(* Logix 5000 project; controller Lab7_1 5069-L306ERM rev 35.16; software revision 35.00 *)

TASK MainTask (continuous, watchdog 500 ms) : MainProgram

MODULES
   Local : 5069-L306ERM (5069 0, rev 35.16)
      IOHub : vendor 1 type 7 code 358 (Ethernet 192.168.110.5, rev 1.1, Output RPI 20 ms)
END_MODULES

PROGRAM MainProgram   (* main routine MainRoutine *)
VAR
   countDown2 : COUNTER := (PRE := 2);
   countDown3 : COUNTER := (PRE := 3);
   counter_0 : COUNTER;
   counter_2 : COUNTER;
   displayTimer : TIMER := (PRE := 5000);
   Dummy : BOOL;
   enable_1_sec : BOOL;
   enable_3_sec : BOOL;
   flash1 : BOOL;
   flash1TOF : TIMER := (PRE := 500);
   flash2 : BOOL;
   flash2TOF : TIMER := (PRE := 1000);
   flash2TON : TIMER := (PRE := 1000);
   flash3 : BOOL;
   flash3TOF : TIMER := (PRE := 1000);
   flash3TON : TIMER := (PRE := 1000);
   flash_1 : BOOL;
   flash_1TOF : TIMER := (PRE := 1000);
   flash_2 : BOOL;
   flash_3 : BOOL;
   HOLD : BOOL;
   HOLD2 : BOOL;
   light_test : BOOL;
   reset : BOOL;
   timer : TIMER := (PRE := 999999999);
   timer_1 : TIMER := (PRE := 1000);
   timer_1_delay : TIMER := (PRE := 1000);
   timer_1_sec : TIMER := (PRE := 1000);
   timer_2 : TIMER := (PRE := 1000);
   timer_2_1 : TIMER := (PRE := 2000);
   timer_2_delay : TIMER := (PRE := 3000, ACC := 2000);
   timer_3_1 : TIMER := (PRE := 3000);
   timer_3_delay : TIMER := (PRE := 5000);
   timer_3_sec : TIMER := (PRE := 1000);
   timer_flash_1 : TIMER := (PRE := 2000);
   timer_flash_2 : TIMER := (PRE := 4000);
   timer_flash_3 : TIMER := (PRE := 6000);
END_VAR

ROUTINE MainRoutine   (* ladder *)
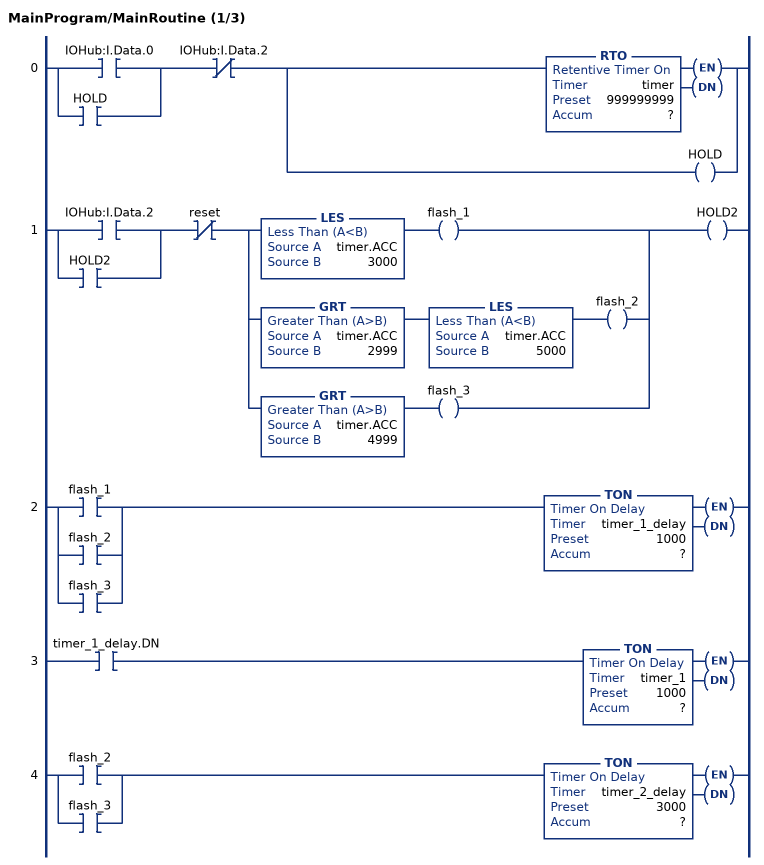
   0: [XIC(IOHub:I.Data.0) ,XIC(HOLD) ]XIO(IOHub:I.Data.2)[RTO(timer,?,?) ,OTE(HOLD) ];
   1: [XIC(IOHub:I.Data.2) ,XIC(HOLD2) ]XIO(reset)[LES(timer.ACC,3000) OTE(flash_1) ,[GRT(timer.ACC,2999) LES(timer.ACC,5000) OTE(flash_2) ,GRT(timer.ACC,4999) OTE(flash_3) ] ]OTE(HOLD2);
   2: [XIC(flash_1) ,XIC(flash_2) ,XIC(flash_3) ]TON(timer_1_delay,?,?);
   3: XIC(timer_1_delay.DN)TON(timer_1,?,?);
   4: [XIC(flash_2) ,XIC(flash_3) ]TON(timer_2_delay,?,?);
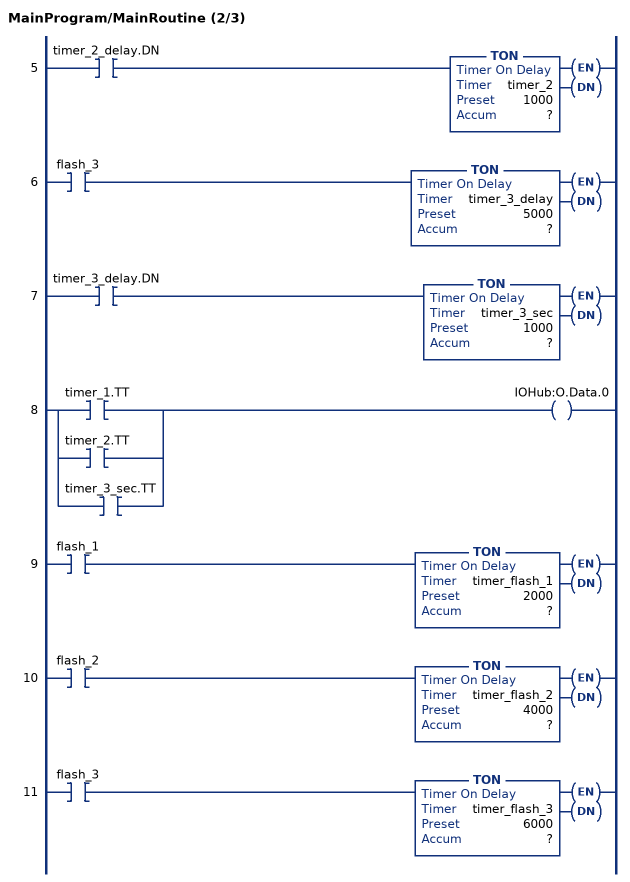
   5: XIC(timer_2_delay.DN)TON(timer_2,?,?);
   6: XIC(flash_3)TON(timer_3_delay,?,?);
   7: XIC(timer_3_delay.DN)TON(timer_3_sec,?,?);
   8: [XIC(timer_1.TT) ,[XIC(timer_2.TT) ,XIC(timer_3_sec.TT) ] ]OTE(IOHub:O.Data.0);
   9: XIC(flash_1)TON(timer_flash_1,?,?);
   10: XIC(flash_2)TON(timer_flash_2,?,?);
   11: XIC(flash_3)TON(timer_flash_3,?,?);
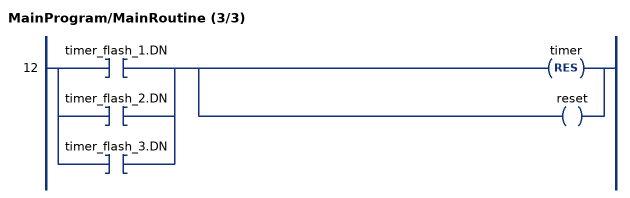
   12: [XIC(timer_flash_1.DN) ,XIC(timer_flash_2.DN) ,XIC(timer_flash_3.DN) ][RES(timer) ,OTE(reset) ];
END_ROUTINE
END_PROGRAM
